TYPE MDP5001_341_O_7CD731EE :
STRUCT
	MDP5001_341_Total_Variant_Value_Out_Index_1_REAL	: UINT;
	MDP5001_341_Total_Variant_Value_Out_Index_2_REAL	: UINT;
	MDP5001_341_Total_Variant_Value_Out_Index_3_REAL	: UINT;
	MDP5001_341_Total_Variant_Value_Out_Index_4_ULINT	: UINT;
	MDP5001_341_Total_Interval_Reset_Interval			: BIT;
END_STRUCT
END_TYPE

(* stored: Version 1.1.0.1, ProductVersion 3.1.4024.12
   DUT MDP5001_341_O_7CD731EE: Id {78232249-ca08-4570-af7f-d20cc69c07ec} *)
